{attribute 'GeneratedUsingTerminal: EPP2339-0003-0016'}
{attribute addProperty BoxType "EPP2339-0003-0016"}
{attribute addProperty Id "OutputAT %Q*ARRAY[0..7] OF BOOL8"}
{attribute addProperty CRC "1253840710"}
{attribute addProperty Size "8"}
TYPE DO_Outputs_Channel_28AC1A9E :
STRUCT
	{attribute addProperty Name "Output"}
	Output AT %Q* : ARRAY[0..7] OF BOOL;
END_STRUCT
END_TYPE

(* stored: Version 1.2.0.0, ProductVersion 3.1.4024.9
   DUT DO_Outputs_Channel_28AC1A9E: Id {228bcb2f-937a-4954-9b6e-6f4d0c870b83} *)
